// TwinCAT 3 PLC project PWFA
// ProgramVersion: 3.1.4024.12
// libraries:
//   Tc2_MC2, * (Beckhoff Automation GmbH)
//   Tc2_NC, * (Beckhoff Automation GmbH)
//   Tc2_Standard, * (Beckhoff Automation GmbH)
//   Tc2_SUPS, * (Beckhoff Automation GmbH)
//   Tc2_System, * (Beckhoff Automation GmbH)
//   Tc2_Utilities, * (Beckhoff Automation GmbH)
//   Tc3_Module, * (Beckhoff Automation GmbH)
// project tree:
//   GVLs/ GVL.TcGVL
//   / PlcTask.TcTTO, RecipeManager.TcRMO (not stored)
//   DUTs/ ST_AxisConfig.TcDUT, ST_AxisIO.TcDUT
//   POUs/ FB_AxisControl.TcPOU, MAIN.TcPOU
//   POUs/PersistentFunction/ FB_Dummy.TcPOU, SLOWTASK.TcPOU, UPSPersitent.TcPOU

CONFIGURATION PWFA
    RESOURCE PLC ON TwinCAT3
        TASK PlcTask(INTERVAL := T#10ms, PRIORITY := 20);
        PROGRAM MAIN WITH PlcTask : MAIN;
    END_RESOURCE
END_CONFIGURATION

// ---- DUTs/ST_AxisConfig.TcDUT
TYPE ST_AxisConfig :
STRUCT
    (* Soft limits *)
    minPosition: REAL;
    maxPosition: REAL;

    (* Motion parameters *)
    targetPosition: REAL;
    targetVelocity: REAL := 0.2;
    jogStep: REAL;

    (* SetPosition *)
    positionSetValue: REAL;

    (* LVDT sensor *)
    lvdtThreshold: REAL;
    lvdtFunctionOn: BOOL := TRUE;
    lvdtManualReleaseAlarm: BOOL;
    scalingFactor_LVDT: REAL := 1;

    (* Position retain (survives power cycle) *)
    currentPositionRetain: REAL;

    (* Axis name for error messages *)
    name: STRING(30);
	
	(* backlash *)
	backlash: REAL:=0.2;          (* mm, 默认 0 *)
	backlashEnable: BOOL;    (* 默认 FALSE *)

END_STRUCT
END_TYPE

// ---- DUTs/ST_AxisIO.TcDUT
TYPE ST_AxisIO :
STRUCT
    (* Limit switches *)
    forwardLimit: BOOL := TRUE;
    forwardLimitSimu: BOOL;
    backwardLimit: BOOL;
    backwardLimitSimu: BOOL;
    touchLimitSwitch: BOOL;

    (* LVDT sensor *)
    lvdtRaw: INT;
	lvdtmA:REAL;
    lvdtScaled: REAL;
    lvdtPV: REAL;
    lvdtOutOfThreshold: BOOL := TRUE;
    lvdtOnceInRangeFlag: INT;

    (* Control buttons (set by HMI or Modbus) *)
    btnMove: BOOL;
    btnJogForward: BOOL;
    btnJogBackward: BOOL;
    btnStop: BOOL;
    btnReset: BOOL;
    btnSetPosition: BOOL;

    (* Status outputs *)
    error: BOOL;
    moving: BOOL;
    moveDone: BOOL;
    positionSetDone: BOOL;
    currentVelocity: REAL;

    (* HMI button interlock outputs *)
    btnJogFwdEnabled: BOOL;
    btnJogBwdEnabled: BOOL;
    btnMoveEnabled: BOOL;
    btnStopEnabled: BOOL;
    btnSetPosEnabled: BOOL;

    (* Internal flags *)
    inputPositionOutOfRange: BOOL;
END_STRUCT
END_TYPE

// ---- GVLs/GVL.TcGVL

{attribute 'qualified_only'}
VAR_GLOBAL CONSTANT
    cMaxAxes : UINT := 10;   (* Change this to add/remove axes without touching code *)
    cActiveAxes : UINT := 10; (* Currently active axes; increase as you add hardware *)
END_VAR

VAR_GLOBAL
    (* ================================================================
       Global control signals
       ================================================================ *)
    simulation: BOOL;
    btn_LocalOrRemote: BOOL := FALSE;
    E_STOP: BOOL; (*急停NC*)
    E_STOP_In AT %I*: BOOL; (*急停NC*)
    E_STOP_rem: BOOL := TRUE; (*远程急停*)
    initStatus: BOOL;

    E_STOP_led: BOOL; (*急停指示*)
    Local_led: BOOL; (*本地模式指示*)
    Remote_led: BOOL; (*远程模式指示*)
    Error: BOOL;
    ErrorId: INT;
    ErrorDescription: STRING;

    (* Plc_EmergencyStop *)
    Plc_EmergencyStop AT %Q*: BOOL := TRUE;
    CabinetEStopRelayTrigged AT %I*: BOOL; (*normal:1,trigged:0*)
    SoftEStopRelayTrigged AT %I*: BOOL; (*normal:1,trigged:0*)

    m_restartTC: BOOL := FALSE;
    E_STOP_ftring: F_TRIG;
    E_STOP_rem_ftring: F_TRIG;

    (* ================================================================
       Axis arrays — add axes by changing cActiveAxes
       ================================================================ *)
    (* NC axis references — link in System Manager *)
    axisRefs: ARRAY[1..cMaxAxes] OF AXIS_REF;

    (* Axis runtime I/O *)
    axesIO: ARRAY[1..cMaxAxes] OF ST_AxisIO;

    (* ================================================================
       Hardware IO — each axis individually mapped in System Manager
       (cannot use arrays because IO addresses may not be sequential)
       ================================================================ *)
    (* Axis 1 HW inputs *)
    forwardLimit_In1 AT %I*: BOOL;
    backwardLimit_In1 AT %I*: BOOL; (*1#电机负向限位.靠近束流*)
    LVDT_In1 AT %I*: INT; (*1#LVDT*)

    (* Axis 2 HW inputs *)
    forwardLimit_In2 AT %I*: BOOL;
    backwardLimit_In2 AT %I*: BOOL;
    LVDT_In2 AT %I*: INT; (*2#LVDT*)

    (* Axis 3-8 HW inputs — uncomment and link as you add axes *)
    forwardLimit_In3 AT %I*: BOOL;
    backwardLimit_In3 AT %I*: BOOL;
    LVDT_In3 AT %I*: INT;

    forwardLimit_In4 AT %I*: BOOL;
    backwardLimit_In4 AT %I*: BOOL;
    LVDT_In4 AT %I*: INT;

    forwardLimit_In5 AT %I*: BOOL;
    backwardLimit_In5 AT %I*: BOOL;
    LVDT_In5 AT %I*: INT;

    forwardLimit_In6 AT %I*: BOOL;
    backwardLimit_In6 AT %I*: BOOL;
    LVDT_In6 AT %I*: INT;

    forwardLimit_In7 AT %I*: BOOL;
    backwardLimit_In7 AT %I*: BOOL;
    LVDT_In7 AT %I*: INT;

    forwardLimit_In8 AT %I*: BOOL;
    backwardLimit_In8 AT %I*: BOOL;
    LVDT_In8 AT %I*: INT;

    (* Axis 9 HW inputs — BL2COL1 *)
    forwardLimit_In9 AT %I*: BOOL;
    backwardLimit_In9 AT %I*: BOOL;
    LVDT_In9 AT %I*: INT;

    (* Axis 10 HW inputs — BL2COL2 *)
    forwardLimit_In10 AT %I*: BOOL;
    backwardLimit_In10 AT %I*: BOOL;
    LVDT_In10 AT %I*: INT;

    (* ================================================================
       All-axis combined commands
       ================================================================ *)
    btn_Move_AxisAll: BOOL;
    RTrig_Move_AxisAll: R_TRIG;
    btn_Stop_AxisAll: BOOL;
    RTrig_Stop_AxisAll: R_TRIG;
    btn_JogForward_AxisAll: BOOL;
    RTrig_JogForward_AxisAll: R_TRIG;
    btn_JogBackward_AxisAll: BOOL;
    RTrig_JogBackward_AxisAll: R_TRIG;
    btn_Reset_AxisAll: BOOL;
    RTrig_Reset_AxisAll: R_TRIG;

    (* ================================================================
       Modbus communication area (EPICS ↔ PLC)
       ================================================================
       Layout:
         Global controls:   %MW0  (1 WORD = 16 bits)
         All-axis commands: %MW2  (1 WORD)
         Per-axis commands: %MW4  (2 WORDs × 10 axes = 20 WORDs)
         Per-axis params:   %MB200 (7 REALs × 10 axes = 70 REALs)
         Per-axis status:   %MW600 (2 WORDs × 10 axes = 20 WORDs)
         Per-axis outputs:  %MB700 (3 REALs × 10 axes = 30 REALs)
         Error info:        %MB820 (INT + STRING)
       ================================================================ *)

    (* ---- EPICS → PLC: Command inputs ---- *)

    (* Global controls — Word 0 (%MW0) *)
    MOD_btn_LocalOrRemote AT %MX0.0: BOOL;
    MOD_btn_E_STOP        AT %MX0.1: BOOL := TRUE;
    MOD_m_restartTC       AT %MX0.2: BOOL;
    (* %MX0.3–%MX0.15 spare *)

    (* All-axis combined commands — Word 1 (%MW2) *)
    MOD_btn_Move_AxisAll        AT %MX2.0: BOOL;
    MOD_btn_JogForward_AxisAll  AT %MX2.1: BOOL;
    MOD_btn_JogBackward_AxisAll AT %MX2.2: BOOL;
    MOD_btn_Stop_AxisAll        AT %MX2.3: BOOL;
    MOD_btn_Reset_AxisAll       AT %MX2.4: BOOL;
    (* %MX2.5–%MX3.7 spare *)

    (* Per-axis BOOL commands — Word 2–17 (%MW4–%MW18)
       Each axis: 1 WORD (8 bits used, 8 spare)
         bit 0: Move      bit 4: Reset
         bit 1: Jog+      bit 5: SetPosition
         bit 2: Jog-      bit 6: LVDT_FunctionOn
         bit 3: Stop      bit 7: LVDT_ManualRelease
       Axis 1 at Word 2 (%MX4.x), Axis N at Word (2+N*2) (%MX(4+(N-1)*4).x)
    *)
    MOD_AxisCmdW AT %MW4: ARRAY[0..19] OF WORD; (* 10 axes × 2 words *)

    (* Per-axis REAL parameters — %MB200, 7 REALs per axis, 10 axes *)
    MOD_AxisParams AT %MB200: ARRAY[0..69] OF REAL;
    (* Layout per axis (28 bytes = 7 REALs):
       [0] targetPosition    [4] minPosition
       [1] targetVelocity    [5] maxPosition
       [2] jogStep           [6] positionSetValue
       [3] lvdtThreshold
    *)

    (* ---- PLC → EPICS: Status outputs ---- *)

    (* Global status — Word 100 (%MW200) *)
   // MOD_E_STOP_led  AT %MX400.0: BOOL;
  //  MOD_Local_led   AT %MX400.1: BOOL;
   // MOD_Remote_led  AT %MX400.2: BOOL;
   // MOD_Error_led   AT %MX400.3: BOOL;
	
    (* Global status LEDs — mapped via MOD_AxisStatW[1] (%MW601) spare word *)
    MOD_E_STOP_led: BOOL;
    MOD_Local_led: BOOL;
    MOD_Remote_led: BOOL;
    MOD_Error_led: BOOL;


    (* Per-axis BOOL status — Word 150–165 (%MW300–%MW330)
       Each axis: 1 WORD (6 bits used, 10 spare)
         bit 0: error          bit 3: backwardLimit
         bit 1: moving         bit 4: moveDone
         bit 2: forwardLimit   bit 5: positionSetDone
    *)
    MOD_AxisStatW AT %MW600: ARRAY[0..19] OF WORD; (* 10 axes × 2 words *)

    (* Per-axis REAL outputs — %MB700, 3 REALs per axis, 10 axes *)
    MOD_AxisOutput AT %MB700: ARRAY[0..29] OF REAL;
    (* Layout per axis (12 bytes = 3 REALs):
       [0] currentVelocity  [1] currentPosition  [2] lvdtPV
    *)

    (* Error info *)
    MOD_ErrorId           AT %MB820: INT;
    MOD_ErrorDescription  AT %MB824: STRING;
END_VAR

VAR_GLOBAL PERSISTENT
    (* Axis configuration — survives TC_Restart and UPS power cycle *)
    axesCfg: ARRAY[1..cMaxAxes] OF ST_AxisConfig;
END_VAR

// ---- POUs/MAIN.TcPOU
PROGRAM MAIN
VAR
    (* Axis FB array — loop over cActiveAxes *)
    fbAxes: ARRAY[1..GVL.cMaxAxes] OF FB_AxisControl;

    (* ============================================================
       Init
       ============================================================ *)
    init_State: INT;
    SetPosition_delay: TON;
    init_delay: TON;
    mcSetPos: ARRAY[1..GVL.cMaxAxes] OF MC_SetPosition;

    (* ============================================================
       All-axis broadcast
       ============================================================ *)
    m_State_AxisAll: INT;
    m_delay: TON;

    (* ============================================================
       Simulation
       ============================================================ *)
    simulation_EStop: BOOL;

    (* ============================================================
       Restart
       ============================================================ *)
    RestartTC: TC_Restart;

    (* ============================================================
       Recipe management
       ============================================================ *)
    RecipeINT: INT;
    RecipeBOOL: BOOL;
    RecipeManCommands: RecipeManCommands;
    SaveParameter: BOOL;
    LoadParameter: BOOL;
    Save_R_TRIG: R_TRIG;
    Read_R_TRIG: R_TRIG;
    loadparameterStatus: INT;
    RecipeBOOL2: BOOL;
    ReturnDwordLoad: DWORD;
    InsertionDeviceName: STRING;
    state_loadParameters: INT;
    LoadRecipeParameters: BOOL;
    loadParametersDone: BOOL;
    CollimatorName: STRING;
    RecipeSavedDate: STRING;
    RecipeDescription: STRING;

    (* ============================================================
       Loop helpers
       ============================================================ *)
    _i: UINT;
    _allDone: BOOL;
END_VAR

(* ============================================================
   MAIN — Storage Ring Collimator (HEPS)
   Multi-axis control with Modbus TCP ↔ EPICS
   ============================================================ *)

(* Copy hardware IO into axis IO structs *)
A_MapHWIO();

(* Initialization — position recovery from persistent memory *)
A_init();

(* Simulation mode — must run BEFORE FB so limit switches are TRUE when MC_Power is called *)
simu();

(* Run all active axis FBs *)
IF GVL.initStatus THEN
    FOR _i := 1 TO GVL.cActiveAxes DO
        fbAxes[_i](
            Axis := GVL.axisRefs[_i],
            IO := GVL.axesIO[_i],
            Cfg := GVL.axesCfg[_i]
        );
    END_FOR
    AxisAll_Motion();
END_IF

(* UPS persistent data *)
UPSPersitent();



(* Modbus data exchange *)
modbus();

(* Restart TC *)
A_RestartTC();

(* Recipe parameters *)
A_InitRecipeParameters();
IF NOT loadParametersDone THEN
    RETURN;
END_IF

ACTION A_init:
(* ============================================================
   Initialization — delay, then restore positions after restart
   axesCfg is VAR_GLOBAL PERSISTENT, so all values survive restart automatically
   ============================================================ *)

(* 3-second startup delay *)
init_delay.PT := T#3S;
init_delay();
init_delay.IN := TRUE;
IF NOT init_delay.Q THEN
    RETURN;
END_IF

(* Call all MC_SetPosition FBs every cycle *)
FOR _i := 1 TO GVL.cActiveAxes DO
    mcSetPos[_i](Axis := GVL.axisRefs[_i]);
END_FOR

SetPosition_delay.PT := T#1S;
SetPosition_delay();

CASE init_State OF
    0:
        (* Wait for all axes to stop *)
        _allDone := TRUE;
        FOR _i := 1 TO GVL.cActiveAxes DO
            IF GVL.axesIO[_i].moving THEN
                _allDone := FALSE;
            END_IF
        END_FOR
        IF _allDone THEN
            init_State := 1;
        END_IF

    1:
        IF NOT GVL.initStatus THEN
            FOR _i := 1 TO GVL.cActiveAxes DO
                mcSetPos[_i].Position := GVL.axesCfg[_i].currentPositionRetain;
                mcSetPos[_i].Execute := TRUE;
            END_FOR
            SetPosition_delay.IN := TRUE;
            init_State := 2;
        END_IF

    2:
        _allDone := TRUE;
        FOR _i := 1 TO GVL.cActiveAxes DO
            IF NOT mcSetPos[_i].Done THEN
                _allDone := FALSE;
            END_IF
        END_FOR
        IF _allDone THEN
            init_State := 88;
        END_IF
        IF SetPosition_delay.Q THEN
            init_State := -100;
        END_IF

    88:
        GVL.initStatus := TRUE;
        FOR _i := 1 TO GVL.cActiveAxes DO
            mcSetPos[_i].Execute := FALSE;
        END_FOR
        SetPosition_delay.IN := FALSE;
        init_State := 0;

    -100:
        GVL.initStatus := FALSE;
        SetPosition_delay.IN := FALSE;
        FOR _i := 1 TO GVL.cActiveAxes DO
            mcSetPos[_i].Execute := FALSE;
        END_FOR
        GVL.Error := TRUE;
        GVL.ErrorId := 1;
        GVL.ErrorDescription := 'init fail';
END_CASE

(* After init, continuously update position retain from NC feedback *)
IF GVL.initStatus THEN
    FOR _i := 1 TO GVL.cActiveAxes DO
        GVL.axesCfg[_i].currentPositionRetain := LREAL_TO_REAL(GVL.axisRefs[_i].NcToPlc.ActPos);
        GVL.axesIO[_i].currentVelocity := LREAL_TO_REAL(GVL.axisRefs[_i].NcToPlc.ActVelo);
    END_FOR
END_IF
END_ACTION

ACTION A_InitRecipeParameters:
CASE state_loadParameters OF
    0:
        LoadParameter := TRUE;
        Read_R_TRIG(CLK := LoadParameter);
        IF Read_R_TRIG.Q THEN
            state_loadParameters := 1;
        END_IF
    1:
        ReturnDwordLoad := RecipeManCommands.LoadAndWriteRecipe(
            RecipeDefinitionName := 'Recipes',
            RecipeName := 'Parameters'
        );
        LoadParameter := FALSE;
        IF ReturnDwordLoad <> 0 THEN
            state_loadParameters := -100;
        ELSE
            LoadRecipeParameters := TRUE;
            LoadParameter := FALSE;
            state_loadParameters := 88;
        END_IF
    88:
        loadParametersDone := TRUE;
    -100:
        loadParametersDone := FALSE;
        GVL.Error := TRUE;
        GVL.ErrorId := 101;
        GVL.ErrorDescription := 'LoadRecipeParameters Error';
END_CASE
END_ACTION

ACTION A_MapHWIO:
(* ============================================================
   Map individual hardware IO variables to axis IO struct arrays
   Must be called every cycle before FB execution
   ============================================================ *)
GVL.axesIO[1].forwardLimit := GVL.forwardLimit_In1;
GVL.axesIO[1].backwardLimit := GVL.backwardLimit_In1;
GVL.axesIO[1].lvdtRaw := GVL.LVDT_In1;

GVL.axesIO[2].forwardLimit := GVL.forwardLimit_In2;
GVL.axesIO[2].backwardLimit := GVL.backwardLimit_In2;
GVL.axesIO[2].lvdtRaw := GVL.LVDT_In2;

GVL.axesIO[3].forwardLimit := GVL.forwardLimit_In3;
GVL.axesIO[3].backwardLimit := GVL.backwardLimit_In3;
GVL.axesIO[3].lvdtRaw := GVL.LVDT_In3;

GVL.axesIO[4].forwardLimit := GVL.forwardLimit_In4;
GVL.axesIO[4].backwardLimit := GVL.backwardLimit_In4;
GVL.axesIO[4].lvdtRaw := GVL.LVDT_In4;

GVL.axesIO[5].forwardLimit := GVL.forwardLimit_In5;
GVL.axesIO[5].backwardLimit := GVL.backwardLimit_In5;
GVL.axesIO[5].lvdtRaw := GVL.LVDT_In5;

GVL.axesIO[6].forwardLimit := GVL.forwardLimit_In6;
GVL.axesIO[6].backwardLimit := GVL.backwardLimit_In6;
GVL.axesIO[6].lvdtRaw := GVL.LVDT_In6;

GVL.axesIO[7].forwardLimit := GVL.forwardLimit_In7;
GVL.axesIO[7].backwardLimit := GVL.backwardLimit_In7;
GVL.axesIO[7].lvdtRaw := GVL.LVDT_In7;

GVL.axesIO[8].forwardLimit := GVL.forwardLimit_In8;
GVL.axesIO[8].backwardLimit := GVL.backwardLimit_In8;
GVL.axesIO[8].lvdtRaw := GVL.LVDT_In8;
END_ACTION

ACTION A_RestartTC:
(* axesCfg is PERSISTENT — survives restart automatically.
   Call FB first so RESTART gets TRUE, then clear both flags. *)
RestartTC(NETID := , RESTART := GVL.m_restartTC, TMOUT := );
IF GVL.m_restartTC THEN
    GVL.m_restartTC := FALSE;
    GVL.MOD_m_restartTC := FALSE;
END_IF
END_ACTION

ACTION AxisAll_Motion:
(* ============================================================
   Broadcast all-axis commands to all active axes
   ============================================================ *)
GVL.RTrig_Move_AxisAll(CLK := GVL.btn_Move_AxisAll);
IF GVL.RTrig_Move_AxisAll.Q THEN
    FOR _i := 1 TO GVL.cActiveAxes DO
        GVL.axesIO[_i].btnMove := TRUE;
    END_FOR
END_IF

GVL.RTrig_Stop_AxisAll(CLK := GVL.btn_Stop_AxisAll);
IF GVL.RTrig_Stop_AxisAll.Q THEN
    FOR _i := 1 TO GVL.cActiveAxes DO
        GVL.axesIO[_i].btnStop := TRUE;
    END_FOR
END_IF

GVL.RTrig_JogForward_AxisAll(CLK := GVL.btn_JogForward_AxisAll);
IF GVL.RTrig_JogForward_AxisAll.Q THEN
    FOR _i := 1 TO GVL.cActiveAxes DO
        GVL.axesIO[_i].btnJogForward := TRUE;
    END_FOR
END_IF

GVL.RTrig_JogBackward_AxisAll(CLK := GVL.btn_JogBackward_AxisAll);
IF GVL.RTrig_JogBackward_AxisAll.Q THEN
    FOR _i := 1 TO GVL.cActiveAxes DO
        GVL.axesIO[_i].btnJogBackward := TRUE;
    END_FOR
END_IF

GVL.RTrig_Reset_AxisAll(CLK := GVL.btn_Reset_AxisAll);
IF GVL.RTrig_Reset_AxisAll.Q THEN
    FOR _i := 1 TO GVL.cActiveAxes DO
        GVL.axesIO[_i].btnReset := TRUE;
    END_FOR
END_IF
END_ACTION

ACTION modbus:
(* ============================================================
   Modbus TCP data exchange (EPICS ↔ PLC)
   ============================================================ *)

(* ---- PLC → EPICS: Status outputs ---- *)

(* Global status *)
GVL.MOD_E_STOP_led := GVL.E_STOP_led;
GVL.MOD_Local_led := GVL.Local_led;
GVL.MOD_Remote_led := GVL.Remote_led;
GVL.MOD_Error_led := GVL.Error;

(* Per-axis status *)
FOR _i := 1 TO GVL.cActiveAxes DO
    (* BOOL status word *)
    GVL.MOD_AxisStatW[(_i-1)*2].0 := GVL.axesIO[_i].error;
    GVL.MOD_AxisStatW[(_i-1)*2].1 := GVL.axesIO[_i].moving;
    GVL.MOD_AxisStatW[(_i-1)*2].2 := GVL.axesIO[_i].forwardLimit;
    GVL.MOD_AxisStatW[(_i-1)*2].3 := GVL.axesIO[_i].backwardLimit;
    GVL.MOD_AxisStatW[(_i-1)*2].4 := GVL.axesIO[_i].moveDone;
    GVL.MOD_AxisStatW[(_i-1)*2].5 := GVL.axesIO[_i].positionSetDone;
    (* bits 6-15 spare *)

    (* REAL outputs *)
    GVL.MOD_AxisOutput[(_i-1)*3 + 0] := GVL.axesIO[_i].currentVelocity;
    GVL.MOD_AxisOutput[(_i-1)*3 + 1] := GVL.axesCfg[_i].currentPositionRetain;
    GVL.MOD_AxisOutput[(_i-1)*3 + 2] := GVL.axesIO[_i].lvdtPV;
END_FOR

(* Error info *)
GVL.MOD_ErrorId := GVL.ErrorId;
GVL.MOD_ErrorDescription := GVL.ErrorDescription;

(* ---- EPICS → PLC: Command inputs ---- *)

(* Local/Remote mode switch *)
IF GVL.btn_LocalOrRemote THEN
    GVL.Local_led := TRUE;
    GVL.Remote_led := FALSE;
ELSE
    GVL.Local_led := FALSE;
    GVL.Remote_led := TRUE;
END_IF

(* restartTC — Remote mode: copy from Modbus; Local mode: set directly by HMI *)
IF GVL.Remote_led THEN
    GVL.m_restartTC := GVL.MOD_m_restartTC;
END_IF

(* Remote mode: read commands from Modbus *)
IF GVL.Remote_led THEN
    (* Global *)
    GVL.E_STOP_rem := GVL.MOD_btn_E_STOP;

    (* All-axis commands from remote *)
    GVL.btn_Move_AxisAll := GVL.MOD_btn_Move_AxisAll;
    GVL.btn_JogForward_AxisAll := GVL.MOD_btn_JogForward_AxisAll;
    GVL.btn_JogBackward_AxisAll := GVL.MOD_btn_JogBackward_AxisAll;
    GVL.btn_Stop_AxisAll := GVL.MOD_btn_Stop_AxisAll;
    GVL.btn_Reset_AxisAll := GVL.MOD_btn_Reset_AxisAll;

    (* Per-axis commands *)
    FOR _i := 1 TO GVL.cActiveAxes DO
        (* BOOL commands *)
        GVL.axesIO[_i].btnMove := GVL.MOD_AxisCmdW[(_i-1)*2].0;
        GVL.axesIO[_i].btnJogForward := GVL.MOD_AxisCmdW[(_i-1)*2].1;
        GVL.axesIO[_i].btnJogBackward := GVL.MOD_AxisCmdW[(_i-1)*2].2;
        GVL.axesIO[_i].btnStop := GVL.MOD_AxisCmdW[(_i-1)*2].3;
        GVL.axesIO[_i].btnReset := GVL.MOD_AxisCmdW[(_i-1)*2].4;
        GVL.axesIO[_i].btnSetPosition := GVL.MOD_AxisCmdW[(_i-1)*2].5;
        GVL.axesCfg[_i].lvdtFunctionOn := GVL.MOD_AxisCmdW[(_i-1)*2].6;
        GVL.axesCfg[_i].lvdtManualReleaseAlarm := GVL.MOD_AxisCmdW[(_i-1)*2].7;

        (* REAL params *)
        GVL.axesCfg[_i].targetPosition := GVL.MOD_AxisParams[(_i-1)*7 + 0];
        GVL.axesCfg[_i].targetVelocity := GVL.MOD_AxisParams[(_i-1)*7 + 1];
        GVL.axesCfg[_i].jogStep := GVL.MOD_AxisParams[(_i-1)*7 + 2];
        GVL.axesCfg[_i].lvdtThreshold := GVL.MOD_AxisParams[(_i-1)*7 + 3];
        GVL.axesCfg[_i].minPosition := GVL.MOD_AxisParams[(_i-1)*7 + 4];
        GVL.axesCfg[_i].maxPosition := GVL.MOD_AxisParams[(_i-1)*7 + 5];
        GVL.axesCfg[_i].positionSetValue := GVL.MOD_AxisParams[(_i-1)*7 + 6];
    END_FOR

    (* All-axis commands override individual when active *)
    IF NOT GVL.MOD_btn_Move_AxisAll THEN
        FOR _i := 1 TO GVL.cActiveAxes DO
            GVL.axesIO[_i].btnMove := GVL.MOD_AxisCmdW[(_i-1)*2].0;
        END_FOR
    ELSE
        GVL.btn_Move_AxisAll := TRUE;
    END_IF
    IF NOT GVL.MOD_btn_Stop_AxisAll THEN
        FOR _i := 1 TO GVL.cActiveAxes DO
            GVL.axesIO[_i].btnStop := GVL.MOD_AxisCmdW[(_i-1)*2].3;
        END_FOR
    ELSE
        GVL.btn_Stop_AxisAll := TRUE;
    END_IF
    IF NOT GVL.MOD_btn_JogForward_AxisAll THEN
        FOR _i := 1 TO GVL.cActiveAxes DO
            GVL.axesIO[_i].btnJogForward := GVL.MOD_AxisCmdW[(_i-1)*2].1;
        END_FOR
    ELSE
        GVL.btn_JogForward_AxisAll := TRUE;
    END_IF
    IF NOT GVL.MOD_btn_JogBackward_AxisAll THEN
        FOR _i := 1 TO GVL.cActiveAxes DO
            GVL.axesIO[_i].btnJogBackward := GVL.MOD_AxisCmdW[(_i-1)*2].2;
        END_FOR
    ELSE
        GVL.btn_JogBackward_AxisAll := TRUE;
    END_IF
    IF NOT GVL.MOD_btn_Reset_AxisAll THEN
        FOR _i := 1 TO GVL.cActiveAxes DO
            GVL.axesIO[_i].btnReset := GVL.MOD_AxisCmdW[(_i-1)*2].4;
        END_FOR
    ELSE
        GVL.btn_Reset_AxisAll := TRUE;
    END_IF
ELSE
    (* Local mode: upload current parameters to Modbus for HMI display *)
    FOR _i := 1 TO GVL.cActiveAxes DO
        GVL.MOD_AxisParams[(_i-1)*7 + 0] := GVL.axesCfg[_i].targetPosition;
        GVL.MOD_AxisParams[(_i-1)*7 + 1] := GVL.axesCfg[_i].targetVelocity;
        GVL.MOD_AxisParams[(_i-1)*7 + 2] := GVL.axesCfg[_i].jogStep;
        GVL.MOD_AxisParams[(_i-1)*7 + 3] := GVL.axesCfg[_i].lvdtThreshold;
        GVL.MOD_AxisParams[(_i-1)*7 + 4] := GVL.axesCfg[_i].minPosition;
        GVL.MOD_AxisParams[(_i-1)*7 + 5] := GVL.axesCfg[_i].maxPosition;
        GVL.MOD_AxisParams[(_i-1)*7 + 6] := GVL.axesCfg[_i].positionSetValue;
    END_FOR
END_IF
END_ACTION

ACTION simu:
(* ============================================================
   Simulation mode — bypass hardware inputs
   ============================================================ *)
IF GVL.simulation THEN
    FOR _i := 1 TO GVL.cActiveAxes DO
        GVL.axesIO[_i].forwardLimit := TRUE;
        GVL.axesIO[_i].backwardLimit := TRUE;
    END_FOR
    GVL.E_STOP := TRUE;
    GVL.E_STOP_led := TRUE;
ELSE
    GVL.E_STOP := GVL.E_STOP_In;
    GVL.E_STOP_led := GVL.E_STOP_In;
    (* Note: limit switch IO is handled in A_MapHWIO before simu *)
END_IF
END_ACTION

END_PROGRAM

// ---- POUs/FB_AxisControl.TcPOU
FUNCTION_BLOCK FB_AxisControl
VAR_IN_OUT
    Axis: AXIS_REF;
    IO: ST_AxisIO;
    Cfg: ST_AxisConfig;
END_VAR
VAR
    (* Motion function blocks *)
    MC_Power: MC_Power;
    MC_MoveAbsolute: MC_MoveAbsolute;
    MC_Jog: MC_Jog;
    MC_Stop: MC_Stop;
    MC_Reset: MC_Reset;
    MC_SetPosition: MC_SetPosition;

    (* State machines *)
    mState: INT;    (* Move absolute state *)
    jState: INT;    (* Jog state *)
    sState: INT;    (* Stop state *)
    rState: INT;    (* Reset state *)
    spState: INT;   (* SetPosition state *)
    esState: INT;   (* E-Stop state *)

    (* Triggers *)
    fTrigReachLS: F_TRIG;
    rTrigEStop: R_TRIG;

    (* Timers *)
    setPosDelay: TON;

    (* Internal flags *)
    mPowerEnable: BOOL;
    mPosProtectionSet: BOOL;
    btnReachLSReset: BOOL;

    (* Shadow copies for FB parameters *)
    mMoveTargetPos: LREAL;
    mMoveTargetVel: LREAL;
    mJogDistance: LREAL;
    mJogVelocity: LREAL;
    mSetPosValue: LREAL;
	
	fTrigJogBackward: F_TRIG;
	fTrigJogForward: F_TRIG;
	
	(* Backlash compensation *)
	backlashPhase: BOOL;
END_VAR

(* ============================================================
   FB_AxisControl — Axis control function block
   Encapsulates: Move, Jog, Stop, Reset, SetPosition,
                 Input protection, E-Stop, LVDT, HMI interlock
   ============================================================ *)

(* ============================================================
   Call all motion FBs every cycle
   (inputs set by state machines below)
   ============================================================ *)
MC_Power(
    Axis := Axis,
    Enable := mPowerEnable,
    Enable_Positive := IO.forwardLimit,
    Enable_Negative := IO.backwardLimit,
    Override := 100
);

MC_MoveAbsolute(
    Axis := Axis,
    Execute := (mState = 3),
    Position := mMoveTargetPos,
    Velocity := mMoveTargetVel
);

MC_Jog(
    Axis := Axis,
    JogForward := (jState = 3 AND IO.btnJogForward AND NOT IO.btnJogBackward),
    JogBackwards := (jState = 3 AND IO.btnJogBackward AND NOT IO.btnJogForward),
    Mode := MC_JOGMODE_INCHING,
    Position := mJogDistance,
    Velocity := mJogVelocity
);

MC_Stop(
    Axis := Axis,
    Execute := (sState = 3)
);

MC_Reset(
    Axis := Axis,
    Execute := (rState = 1)
);

setPosDelay.PT := T#0.1S;
setPosDelay();

MC_SetPosition(
    Axis := Axis,
    Execute := (spState = 2),
    Position := mSetPosValue
);

(* ============================================================
   Input position protection
   ============================================================ *)
IF IO.btnMove THEN
    IF Cfg.targetPosition >= Cfg.minPosition AND Cfg.targetPosition <= Cfg.maxPosition THEN
        IO.inputPositionOutOfRange := FALSE;
        GVL.Error := FALSE;
        GVL.ErrorId := 0;
        GVL.ErrorDescription := '';
    ELSE
        IO.inputPositionOutOfRange := TRUE;
        GVL.Error := TRUE;
        GVL.ErrorId := 1001;
        GVL.ErrorDescription := CONCAT(Cfg.name, '_InputPositionOutOfRange');
        RETURN;
    END_IF
END_IF

(* ============================================================
   Running status
   ============================================================ *)
Axis.ReadStatus();
IO.moving := Axis.Status.Moving;

(* Error status from NC *)
IF Axis.NcToPlc.ErrorCode = 0 THEN
    IO.error := FALSE;
ELSE
    IO.error := TRUE;
    GVL.Error := TRUE;
    GVL.ErrorId := 1002;
    GVL.ErrorDescription := CONCAT(Cfg.name, '.NcToPlc.ErrorCode<>0');
END_IF

(* Move done *)
IO.moveDone := MC_MoveAbsolute.Done OR MC_Jog.Done;

(* ============================================================
   Power enable logic — on if any motion state is active
   ============================================================ *)
mPowerEnable := (mState >= 1 AND mState <> 88 AND mState <> -100)
             OR (jState >= 1 AND jState <> 88 AND jState <> -100)
             OR (sState >= 1 AND sState <> 88 AND sState <> -100);

(* ============================================================
   Position Move state machine
   ============================================================ *)
CASE mState OF
    0:
        IF NOT IO.error THEN
            mState := 1;
        ELSE
            mState := -100;
        END_IF
    1:
        IF NOT MC_Power.Status THEN
            (* power is enabled via mPowerEnable above *)
        ELSE
            mState := 2;
        END_IF
    2:
        mMoveTargetVel := Cfg.targetVelocity;
        IF IO.btnMove THEN
            (* backlash: reverse move → compensate first *)
            IF Cfg.backlashEnable
               AND (Cfg.backlash > 0.0)
               AND (Cfg.targetPosition < Cfg.currentPositionRetain) THEN
                mMoveTargetPos := Cfg.targetPosition - Cfg.backlash;
                backlashPhase := TRUE;
            ELSE
                mMoveTargetPos := Cfg.targetPosition;
                backlashPhase := FALSE;
            END_IF
            mState := 3;
        END_IF
    3:
        IF MC_MoveAbsolute.Done THEN
            IF backlashPhase THEN
                (* backlash pass complete → load final target *)
                mMoveTargetPos := Cfg.targetPosition;
                backlashPhase := FALSE;
                mState := 10;
            ELSE
                mState := 88;
            END_IF
        END_IF
    10:
        mState := 3;    (* re-trigger Execute rising edge *)
    88:
        IO.btnMove := FALSE;
        mState := 0;
    -100:
        IO.btnMove := FALSE;
        GVL.Error := TRUE;
        IO.error := TRUE;
        GVL.ErrorId := 1002;
        GVL.ErrorDescription := CONCAT(Cfg.name, '_move_error');
END_CASE

(* ============================================================
   Jog state machine
   ============================================================ *)
CASE jState OF
    0:
        IF NOT IO.error THEN
            jState := 1;
        ELSE
            jState := -100;
        END_IF
    1:
        IF NOT MC_Power.Status THEN
            (* waiting for power *)
        ELSE
            jState := 2;
        END_IF
    2:
        mJogDistance := Cfg.jogStep;
        mJogVelocity := Cfg.targetVelocity;
		
		IF IO.btnJogForward AND NOT IO.btnJogBackward THEN
			IF Cfg.currentPositionRetain + Cfg.jogStep <= Cfg.maxPosition THEN
				GVL.Error := FALSE;
				GVL.ErrorId := 0;
				jState := 3;
			ELSE
				IO.btnJogForward := FALSE;          // ← 立即清按钮，防 Modbus 重写
				GVL.Error := TRUE;
				GVL.ErrorId := 1002;
				GVL.ErrorDescription := CONCAT('exceed ', CONCAT(Cfg.name, '_maxPosition'));
			END_IF
		END_IF
		
		IF IO.btnJogBackward AND NOT IO.btnJogForward THEN
			IF Cfg.currentPositionRetain - Cfg.jogStep >= Cfg.minPosition THEN
				GVL.Error := FALSE;
				GVL.ErrorId := 0;
				jState := 3;
			ELSE
				IO.btnJogBackward := FALSE;         // ← 同上
				GVL.Error := TRUE;
				GVL.ErrorId := 1003;
				GVL.ErrorDescription := CONCAT('less than ', CONCAT(Cfg.name, '_minPosition'));
			END_IF
		END_IF
	
    3:
        (* Buttons kept TRUE so MC_Jog sees them next cycle; cleared in state 88/-100 *)
        IF MC_Jog.Error THEN
            jState := -100;
        ELSIF MC_Jog.Done THEN
            jState := 88;
        END_IF
    88:
        IO.btnJogForward := FALSE;
        IO.btnJogBackward := FALSE;
        jState := 0;
    -100:
        IO.btnJogForward := FALSE;
        IO.btnJogBackward := FALSE;
        GVL.Error := TRUE;
        IO.error := TRUE;
        GVL.ErrorId := 1002;
        GVL.ErrorDescription := CONCAT(Cfg.name, '_jog_error');
END_CASE

(* ============================================================
   Stop state machine
   ============================================================ *)
CASE sState OF
    0:
        sState := 1;
    1:
        IF NOT MC_Power.Status THEN
            (* waiting for power *)
        ELSE
            sState := 2;
        END_IF
    2:
        IF IO.btnStop THEN
            sState := 3;
        END_IF
    3:
        IF MC_Stop.Done THEN
            sState := 88;
        END_IF
    88:
        IO.btnStop := FALSE;
        sState := 0;
        (* Reset all other states on stop *)
        IO.btnMove := FALSE;
        IO.btnJogForward := FALSE;
        IO.btnJogBackward := FALSE;
        mState := 0;
        jState := 0;
    -100:
        IO.btnStop := FALSE;
        GVL.Error := TRUE;
        IO.error := TRUE;
        GVL.ErrorId := 1002;
        GVL.ErrorDescription := CONCAT(Cfg.name, '_stop_error');
        IO.btnMove := FALSE;
        IO.btnJogForward := FALSE;
        IO.btnJogBackward := FALSE;
        mState := 0;
        jState := 0;
END_CASE

(* ============================================================
   Reset state machine
   ============================================================ *)
CASE rState OF
    0:
        IF IO.btnReset OR btnReachLSReset THEN
            rState := 1;
        END_IF
    1:
        IF MC_Reset.Done THEN
            rState := 88;
        END_IF
    88:
        rState := 0;
        IO.btnReset := FALSE;
        btnReachLSReset := FALSE;
        (* Reset all other states *)
        IO.btnMove := FALSE;
        IO.btnJogForward := FALSE;
        IO.btnJogBackward := FALSE;
        mState := 0;
        sState := 0;
        jState := 0;
END_CASE

(* ============================================================
   SetPosition state machine
   ============================================================ *)
IF IO.btnSetPosition THEN
    CASE spState OF
        0:
            IF NOT IO.moving THEN
                spState := 1;
            END_IF
        1:
            mSetPosValue := Cfg.positionSetValue;
            setPosDelay.IN := TRUE;
            spState := 2;
        2:
            IF MC_SetPosition.Done THEN
                spState := 88;
            END_IF
            IF setPosDelay.Q THEN
                spState := -100;
            END_IF
        88:
            IO.positionSetDone := TRUE;
            setPosDelay.IN := FALSE;
            spState := 0;
            IO.btnSetPosition := FALSE;
        -100:
            IO.positionSetDone := FALSE;
            setPosDelay.IN := FALSE;
            IO.btnSetPosition := FALSE;
            spState := 0;
    END_CASE
ELSE
    setPosDelay.IN := FALSE;
END_IF

IF NOT IO.btnSetPosition THEN
    IO.positionSetDone := FALSE;
END_IF
(* ============================================================
   Emergency stop handler
   ============================================================ *)
IF NOT(GVL.E_STOP AND GVL.E_STOP_rem AND GVL.Plc_EmergencyStop) THEN
    CASE esState OF
        0:
            esState := 1;
        1:
            GVL.E_STOP_led := FALSE;
            mPowerEnable := FALSE;
            IO.btnStop := TRUE;
            GVL.Error := TRUE;
            GVL.ErrorId := 101;
            GVL.ErrorDescription := 'E_STOP';
    END_CASE
END_IF

rTrigEStop(CLK := GVL.E_STOP AND GVL.E_STOP_rem AND GVL.Plc_EmergencyStop);
IF rTrigEStop.Q THEN
    GVL.E_STOP_led := TRUE;
    GVL.Error := FALSE;
    GVL.ErrorId := 0;
    GVL.ErrorDescription := '';
    esState := 0;
END_IF

(* ============================================================
   Limit switch auto-reset (both limits hit -> trigger reset)
   ============================================================ *)
IO.touchLimitSwitch := IO.forwardLimit AND IO.backwardLimit;

fTrigReachLS(CLK := IO.forwardLimit AND IO.backwardLimit);
IF fTrigReachLS.Q THEN
    IO.btnReset := TRUE;
    btnReachLSReset := TRUE;
END_IF

(* ============================================================
   LVDT sensor processing
   ============================================================ *)
//raw data convert mA
IO.lvdtmA:=(INT_TO_REAL(IO.lvdtRaw)/32767)*16+4;
//mA convert to actual position:4-20mA → -10~40mm
IO.lvdtPV:= ((IO.lvdtmA-4.0)/16.0)*50.0-10;

IF Cfg.lvdtFunctionOn THEN
    IF IO.lvdtPV <= Cfg.lvdtThreshold THEN
        IO.lvdtOutOfThreshold := FALSE;
        GVL.Error := TRUE;
        GVL.ErrorDescription := CONCAT(Cfg.name, '_LVDT In Alarm Range');
        IO.lvdtOnceInRangeFlag := 1;
    END_IF
    IF IO.lvdtOnceInRangeFlag = 1 THEN
        IO.lvdtOutOfThreshold := FALSE;
        GVL.Error := TRUE;
        GVL.ErrorDescription := CONCAT(Cfg.name, '_LVDT In Alarm Range');
        IF Cfg.lvdtManualReleaseAlarm THEN
            GVL.Error := FALSE;
            GVL.ErrorDescription := '';
            IO.lvdtOnceInRangeFlag := 0;
            Cfg.lvdtManualReleaseAlarm := FALSE;
            IO.lvdtOutOfThreshold := TRUE;
        END_IF
    END_IF
END_IF

(* ============================================================
   HMI button interlock logic (Local mode only)
   ============================================================ *)
(* JOG+ enabled? *)
IF IO.forwardLimit AND GVL.E_STOP AND GVL.Local_led AND NOT IO.error
   AND NOT IO.moving AND NOT IO.btnMove AND NOT IO.btnJogBackward THEN
    IO.btnJogFwdEnabled := TRUE;
ELSE
    IO.btnJogFwdEnabled := FALSE;
END_IF

(* JOG- enabled? *)
IF IO.backwardLimit AND GVL.E_STOP AND GVL.Local_led AND NOT IO.error
   AND NOT IO.moving AND NOT IO.btnMove AND NOT IO.btnJogForward THEN
    IO.btnJogBwdEnabled := TRUE;
ELSE
    IO.btnJogBwdEnabled := FALSE;
END_IF

(* Position Move enabled? *)
IF GVL.E_STOP AND GVL.Local_led AND NOT IO.error AND NOT IO.moving
   AND NOT IO.btnJogForward AND NOT IO.btnJogBackward THEN
    IO.btnMoveEnabled := TRUE;
ELSE
    IO.btnMoveEnabled := FALSE;
END_IF

(* SetPosition enabled? *)
IF GVL.E_STOP AND GVL.Local_led AND NOT IO.error AND NOT IO.moving THEN
    IO.btnSetPosEnabled := TRUE;
ELSE
    IO.btnSetPosEnabled := FALSE;
END_IF

(* Stop enabled? *)
IF GVL.E_STOP AND GVL.Local_led AND NOT IO.error THEN
    IO.btnStopEnabled := TRUE;
ELSE
    IO.btnStopEnabled := FALSE;
END_IF

END_FUNCTION_BLOCK

// ---- POUs/PersistentFunction/UPSPersitent.TcPOU
PROGRAM UPSPersitent
VAR
		 
	 (* UPS related ... *)
	fbUPS			: FB_S_UPS_CX51x0;			(* UPS-FB instance *)
					(* Default Values of FB_S_UPS_CX51x0-Inputs:
						sNetID 			:= '' ==> local netid
						iPLCPort 		:= AMSPORT_R0_PLC_RTS1 ==> 801 = 1st Runtime System
						iUPSPort		:= 16#588 ==> Port for reading Power State of UPS
						tTimeout 		:= DEFAULT_ADS_TIMEOUT ==> 5S
						eUpsMode 		:= eSUPS_WrPersistData_Shutdown ==> writing persistent data + shutdown
						ePersistentMode := SPDM_2PASS ==> All data is from same plc cycle, cycletime exceeds possible. Plc stops with the shutdown, a few cycles after writing persistent data. 
						tRecoverTime 	:= T#10s ==> 10s power to recover from short power failure before eSUPS_PowerOK is reported (in mode eSUPS_WrPersistData_NoShutdown/eSUPS_CheckPowerStatus)
					*)
	eUpsMode		: E_S_UPS_Mode	:= eSUPS_WrPersistData_Shutdown; (* UPS mode (writing persistent data + shutdown) *)

	(* !!! TO DO: REPLACE WITH YOUR PLC VARIABLES/FB INSTANCES !!! regular PLC variables/FB instances ... *)
	iCounter		: UDINT;					(* non persistent counter *)
	fbMachineFast	: FB_Dummy;					(* demo fb instance *)
END_VAR
VAR PERSISTENT
	(* !!! TO DO: REPLACE WITH YOUR PERSISTENT PLC VARIABLES !!! persistent variables ... *)
	iCounter_P				: UDINT;			(* persistent counter *)
	iPowerFailureCounter_P	: UDINT;			(* persistent counter of power failures *)
END_VAR

(* S-UPS Demo *)

(* call UPS-FB instance in first lines of the fastest PLC Task *)
fbUPS(eUpsMode := eUpsMode);
(* eUpsMode =							in case of powerfailure:
	 eSUPS_WrPersistData_Shutdown 		 	writing of persistent data + shutdown
	 eSUPS_WrPersistData_NoShutdown 		writing of PERSISTENT data, no shutdown
	 eSUPS_CheckPowerStatus 				reports powerfailure without ACTION (no writing, no shutdown) 
	 eSUPS_ImmediateShutdown 				skips writing of data, immediate shutdown
*)

(* evaluate UPS State *)
IF eGlobalSUpsState = eSUPS_PowerFailure THEN
	(* first cycle of powerfailure *)

	(* execute code that should only be done once with each powerfailure, i.e. increase powerfailure counter *)
	iPowerFailureCounter_P := iPowerFailureCounter_P + 1;
ELSIF eGlobalSUpsState > eSUPS_PowerFailure THEN
	(* next cycles of powerfailure *)

	(* skip regular code execution for the remaining cycles of the powerfailure/writing of persistent data/quick shutdown  ... *)
	RETURN;
END_IF


(* !!! TO DO: REPLACE WITH YOUR PLC CODE !!! regular code execution *)
iCounter := iCounter + 1;
iCounter_P := iCounter_P + 1;

fbMachineFast();

END_PROGRAM

// ---- POUs/PersistentFunction/FB_Dummy.TcPOU
FUNCTION_BLOCK FB_Dummy
VAR_INPUT
END_VAR
VAR_OUTPUT
END_VAR
VAR
	(* not persistent variables ... *)
	iCounter		: UDINT;			(* non persistent counter *)
END_VAR
VAR PERSISTENT
	(* persistent variables ... *)
	iCounter_P		: UDINT;			(* persistent counter *)
END_VAR

iCounter 	:= iCounter + 1;
iCounter_P	:= iCounter_P + 1;

END_FUNCTION_BLOCK

// ---- POUs/PersistentFunction/SLOWTASK.TcPOU
PROGRAM SLOWTASK
VAR
	(* !!! TO DO: REPLACE WITH YOUR PLC VARIABLES/FB INSTANCES !!! regular PLC variables/FB instances ... *)
	iCounter			: UDINT;					(* non persistent counter *)
	fbMachineSlow		: FB_Dummy;					(* demo fb instance *)
END_VAR
VAR PERSISTENT
	(* !!! TO DO: REPLACE WITH YOUR PERSISTENT PLC VARIABLES !!! persistent variables ... *)
	iCounter_P				: UDINT;			(* persistent counter *)
END_VAR

(* evaluate UPS State *)
IF eGlobalSUpsState > eSUPS_PowerFailure THEN
	(* next cycles of powerfailure *)

	(* skip regular code execution for the remaining cycles of the powerfailure/writing of persistent data/quick shutdown  ... *)
	RETURN;
END_IF


(* !!! TO DO: REPLACE WITH YOUR PLC CODE !!! regular code execution *)
iCounter := iCounter + 1;
iCounter_P := iCounter_P + 1;
fbMachineSlow();

END_PROGRAM
